# EPICS substitutions: db/music_adc_ch.substitutions
###############################################################################
#
# MUSIC ADC channel definitions
#
# Hardware:
#     mesytec MDPP-32-PADC
#
# Authors:
#     i.keshelashvili@gsi.de
#
###############################################################################

global
{
    P = SFRS
}

file "db/music_adc_ch.template"
{
    pattern
    {
        CHAMBER, FILD_CAGE, CHANNEL
    }

    # FMF1 MUSIC field cage 1
    { FMF1, 1, 01 }
    { FMF1, 1, 02 }
    { FMF1, 1, 03 }
    { FMF1, 1, 04 }
    { FMF1, 1, 05 }
    { FMF1, 1, 06 }
    { FMF1, 1, 07 }
    { FMF1, 1, 08 }
    { FMF1, 1, 09 }
    { FMF1, 1, 10 }
    { FMF1, 1, 11 }
    { FMF1, 1, 12 }
    { FMF1, 1, 13 }
    { FMF1, 1, 14 }
    { FMF1, 1, 15 }
    { FMF1, 1, 16 }
    { FMF1, 1, 17 }
    { FMF1, 1, 18 }
    { FMF1, 1, 19 }
    { FMF1, 1, 20 }
    { FMF1, 1, 21 }
    { FMF1, 1, 22 }
    { FMF1, 1, 23 }
    { FMF1, 1, 24 }
    { FMF1, 1, 25 }
    { FMF1, 1, 26 }
    { FMF1, 1, 27 }
    { FMF1, 1, 28 }
    { FMF1, 1, 29 }
    { FMF1, 1, 30 }
    { FMF1, 1, 31 }
    { FMF1, 1, 32 }

    # FMF1 MUSIC field cage 2
    { FMF1, 2, 01 }
    { FMF1, 2, 02 }
    { FMF1, 2, 03 }
    { FMF1, 2, 04 }
    { FMF1, 2, 05 }
    { FMF1, 2, 06 }
    { FMF1, 2, 07 }
    { FMF1, 2, 08 }
    { FMF1, 2, 09 }
    { FMF1, 2, 10 }
    { FMF1, 2, 11 }
    { FMF1, 2, 12 }
    { FMF1, 2, 13 }
    { FMF1, 2, 14 }
    { FMF1, 2, 15 }
    { FMF1, 2, 16 }
    { FMF1, 2, 17 }
    { FMF1, 2, 18 }
    { FMF1, 2, 19 }
    { FMF1, 2, 20 }
    { FMF1, 2, 21 }
    { FMF1, 2, 22 }
    { FMF1, 2, 23 }
    { FMF1, 2, 24 }
    { FMF1, 2, 25 }
    { FMF1, 2, 26 }
    { FMF1, 2, 27 }
    { FMF1, 2, 28 }
    { FMF1, 2, 29 }
    { FMF1, 2, 30 }
    { FMF1, 2, 31 }
    { FMF1, 2, 32 }

    # FHF1 MUSIC field cage 1
    { FHF1, 1, 01 }
    { FHF1, 1, 02 }
    { FHF1, 1, 03 }
    { FHF1, 1, 04 }
    { FHF1, 1, 05 }
    { FHF1, 1, 06 }
    { FHF1, 1, 07 }
    { FHF1, 1, 08 }
    { FHF1, 1, 09 }
    { FHF1, 1, 10 }
    { FHF1, 1, 11 }
    { FHF1, 1, 12 }
    { FHF1, 1, 13 }
    { FHF1, 1, 14 }
    { FHF1, 1, 15 }
    { FHF1, 1, 16 }
    { FHF1, 1, 17 }
    { FHF1, 1, 18 }
    { FHF1, 1, 19 }
    { FHF1, 1, 20 }
    { FHF1, 1, 21 }
    { FHF1, 1, 22 }
    { FHF1, 1, 23 }
    { FHF1, 1, 24 }
    { FHF1, 1, 25 }
    { FHF1, 1, 26 }
    { FHF1, 1, 27 }
    { FHF1, 1, 28 }
    { FHF1, 1, 29 }
    { FHF1, 1, 30 }
    { FHF1, 1, 31 }
    { FHF1, 1, 32 }

    # FHF1 MUSIC field cage 2
    { FHF1, 2, 01 }
    { FHF1, 2, 02 }
    { FHF1, 2, 03 }
    { FHF1, 2, 04 }
    { FHF1, 2, 05 }
    { FHF1, 2, 06 }
    { FHF1, 2, 07 }
    { FHF1, 2, 08 }
    { FHF1, 2, 09 }
    { FHF1, 2, 10 }
    { FHF1, 2, 11 }
    { FHF1, 2, 12 }
    { FHF1, 2, 13 }
    { FHF1, 2, 14 }
    { FHF1, 2, 15 }
    { FHF1, 2, 16 }
    { FHF1, 2, 17 }
    { FHF1, 2, 18 }
    { FHF1, 2, 19 }
    { FHF1, 2, 20 }
    { FHF1, 2, 21 }
    { FHF1, 2, 22 }
    { FHF1, 2, 23 }
    { FHF1, 2, 24 }
    { FHF1, 2, 25 }
    { FHF1, 2, 26 }
    { FHF1, 2, 27 }
    { FHF1, 2, 28 }
    { FHF1, 2, 29 }
    { FHF1, 2, 30 }
    { FHF1, 2, 31 }
    { FHF1, 2, 32 }

    # FHF1 MUSIC field cage 3
    { FHF1, 3, 01 }
    { FHF1, 3, 02 }
    { FHF1, 3, 03 }
    { FHF1, 3, 04 }
    { FHF1, 3, 05 }
    { FHF1, 3, 06 }
    { FHF1, 3, 07 }
    { FHF1, 3, 08 }
    { FHF1, 3, 09 }
    { FHF1, 3, 10 }
    { FHF1, 3, 11 }
    { FHF1, 3, 12 }
    { FHF1, 3, 13 }
    { FHF1, 3, 14 }
    { FHF1, 3, 15 }
    { FHF1, 3, 16 }
    { FHF1, 3, 17 }
    { FHF1, 3, 18 }
    { FHF1, 3, 19 }
    { FHF1, 3, 20 }
    { FHF1, 3, 21 }
    { FHF1, 3, 22 }
    { FHF1, 3, 23 }
    { FHF1, 3, 24 }
    { FHF1, 3, 25 }
    { FHF1, 3, 26 }
    { FHF1, 3, 27 }
    { FHF1, 3, 28 }
    { FHF1, 3, 29 }
    { FHF1, 3, 30 }
    { FHF1, 3, 31 }
    { FHF1, 3, 32 }
}
